DATA_BLOCK "JAMB_CLEANER_DB"	// DB 8
AUTHOR : Kamillas
VERSION : 0.1
  STRUCT
   JC_CAR_TRA_FWD_LS : BOOL ;	//JAMB CLEANER CARRIAGE TRAVEL FORWARD LIMIT SWITCH
   JC_CAR_TRA_RET_LS : BOOL ;	//JAMB CLEANER CARRIAGE TRAVEL RETRACT LIMIT SWITCH
   JC_VER_CLNR_UP_LS : BOOL ;	//JAMB CLEANER VERTICAL CLEANER UP LIMIT SWITCH
   JC_VER_CLNR_DN_LS : BOOL ;	//JAMB CLEANER VERTICAL CLEANER DOWN LIMIT SWITCH
   JC_VER_CLNR_HME_LS : BOOL ;	//JAMB CLEANER VERTICAL CLEANER HOME LIMIT SWITCH
   JC_CRA_TRA_FWD_STA_PB : BOOL ;	//JAMB CLEANER CARRIAGE TRAVEL FORWARD PUSH BUTTON
   JC_CRA_TRA_RET_STA_PB : BOOL ;	//JAMB CLEANER CARRIAGE TRAVEL RETRACT PUSH BUTTON
   JC_VC_UP_STA_PB : BOOL ;	//JAMB CLEANER VERTICAL CLEANER UP START PUSH BUTTON
   JC_VC_DN_STA_PB : BOOL ;	//JAMB CLEANER VERTICAL CLEANER DOWN START PUSH BUTTON
   JC_STP_PB : BOOL ;	//JAMB CLEANER OPERATIONS STOP PUSH BUTTON
   JC_VC_HME_STA_PB : BOOL ;	//JAMB CLEANER VERTICAL CLEANER HOME START PUSH BUTTON
   JC_CAR_TRA_FWD_CMD : BOOL ;	//JAMB CLEANER CARRIAGE TRAVEL FORWARD COMMAND
   JC_CAR_TRA_RET_CMD : BOOL ;	//JAMB CLEANER CARRIAGE TRAVEL RETRACT COMMAND
   JC_VC_UP_CMD : BOOL ;	//JAMB CLEANER VERTICAL CLEANER UP COMMAND
   JC_VC_DN_CMD : BOOL ;	//JAMB CLEANER VERTICAL CLEANER DOWN COMMAND
   JC_CAR_TRA_FWD_IND : BOOL ;	//JAMB CLEANER CARRIAGE TRAVEL FORWARD INDICATOR
   JC_CAR_TRA_RET_IND : BOOL ;	//JAMB CLEANER CARRIAGE TRAVEL RETRACT INDICATOR
   JC_VC_UP_IND : BOOL ;	//JAMB CLEANER VERTICAL CLEANER UP INDICATOR
   JC_VC_DN_IND : BOOL ;	//JAMB CLEANER VERTICAL CLEANER DOWN INDICATOR
   JC_VC_HME_IND : BOOL ;	//JAMB CLEANER VERTICAL CLEANER HOME INDIATOR
   CLN_OVN_JMB_STA_PB : BOOL ;	//CLEAN OVEN JAMB AUTO START PUSH BUTTON
   CLN_OVN_JMB_STP_PB : BOOL ;	//CLEAN OVEN JAMB AUTO STOP PUSH BUTTON
   CLN_OVN_JMB_IND : BOOL ;	//CLEAN OVEN JAMB AUTO INDICATOR
   JC_TRA_FWD_OP_CUT : BOOL ;	//JAMB CLEANER TRAVEL FORWARD OUTPUT CUT
   JC_TRA_FWD_OP_CUT_TMR : INT ;	//JAMB CLEANER TRAVEL FORWARD OUTPUT CUT TIMER
   JC_TRA_AUTO_FWD_OVR : BOOL ;	//JAMB CLEANER TRAVEL AUTO FORWARD OVER
   JC_TRA_AUTO_FWD_DEL : INT  := 3;	//JAMB CLEANER TRAVEL AUTO FORWARD OVER DELAY
   JC_TRA_AUTO_FWD_DEL_TMR : INT ;	//JAMB CLEANER TRAVEL AUTO FORWARD OVER DELAY TIMER
   JC_TRA_AUTO_FWD_SET : BOOL ;	//JAMB CLEANER AUTO TRAVEL FORWARD SET
   JC_TRA_RET_OP_CUT : BOOL ;	//JAMB CLEANER TRAVEL RETRACT OUTPUT CUT
   JC_TRA_RET_OP_CUT_TMR : INT ;	//JAMB CLEANER TRAVEL RETRACT OUTPUT CUT TIMER
   JC_TRA_AUTO_RET_OVR : BOOL ;	//JAMB CLEANER TRAVEL AUTO RETRACT OVER
   JC_TRA_AUTO_RET_DEL : INT  := 3;	//JAMB CLEANER TRAVEL AUTO RETRACT OVER DELAY
   JC_TRA_AUTO_RET_DEL_TMR : INT ;	//JAMB CLEANER TRAVEL AUTO RETRACT OVER DELAY TIMER
   JC_TRA_AUTO_RET_SET : BOOL ;	//JAMB CLEANER AUTO TRAVEL RETRACT SET
   JC_VC_FWD_OP_CUT : BOOL ;	//JAMB CLEANER VERTICAL CLEANER FORWARD OUTPUT CUT
   JC_VC_FWD_OP_CUT_TMR : INT ;	//JAMB CLEANER VERTICAL CLEANER FORWARD OUTPUT CUT TIMER
   JC_VC_AUTO_FWD_OVR : BOOL ;	//JAMB CLEANER VERTICAL CLEANER AUTO FORWARD OVER
   JC_VC_AUTO_FWD_DEL : INT  := 3;	//JAMB CLEANER VERTICAL CLEANER AUTO FORWARD OVER DELAY
   JC_VC_AUTO_FWD_DEL_TMR : INT ;	//JAMB CLEANER VERTICAL CLEANER AUTO FORWARD OVER DELAY TIMER
   JC_VC_AUTO_FWD_SET : BOOL ;	//JAMB CLEANER AUTO VERTICAL CLEANER FORWARD SET
   JC_VC_RET_OP_CUT : BOOL ;	//JAMB CLEANER VERTICAL CLEANER RETRACT OUTPUT CUT
   JC_VC_RET_OP_CUT_TMR : INT ;	//JAMB CLEANER VERTICAL CLEANER RETRACT OUTPUT CUT TIMER
   JC_VC_AUTO_RET_OVR : BOOL ;	//JAMB CLEANER VERTICAL CLEANER AUTO RETRACT OVER
   JC_VC_AUTO_RET_DEL : INT  := 3;	//JAMB CLEANER VERTICAL CLEANER AUTO RETRACT OVER DELAY
   JC_VC_AUTO_RET_DEL_TMR : INT ;	//JAMB CLEANER VERTICAL CLEANER AUTO RETRACT OVER DELAY TIMER
   JC_VC_AUTO_RET_SET : BOOL ;	//JAMB CLEANER AUTO VERTICAL CLEANER RETRACT SET
   JC_AUTO_SS : BOOL ;	//JAMB CLEANER AUTO MODE SELECTOR SWITCH
   JC_MAN_SS : BOOL ;	//JAMB CLEANER MANUAL MODE SELECTOR SWITCH
   JC_LOC_SS : BOOL ;	//JAMB CLEANER LOCAL MODE SELECTOR SWITCH
   JC_AUTO_STA_PB : BOOL ;	//JAMB CLEANER AUTO START PUSH BUTTON
   JC_ILK_BIT : BOOL ;	//JAMB CLEANER INTERLOCK BIT
   PULSE_1 : BOOL ;	//PULSE 1
   PULSE_2 : BOOL ;	//PULSE 2
   PULSE_3 : BOOL ;	//PULSE 3
   PULSE_4 : BOOL ;	//PULSE 4
   PULSE_5 : BOOL ;	//PULSE 5
   PULSE_6 : BOOL ;	//PULSE 6
   PULSE_7 : BOOL ;	//PULSE 7
   PULSE_8 : BOOL ;	//PULSE 8
   PULSE_9 : BOOL ;	//PULSE 9
   PULSE_10 : BOOL ;	//PULSE 10
   PULSE_11 : BOOL ;	//PULSE 11
   PULSE_12 : BOOL ;	//PULSE 12
   PULSE_13 : BOOL ;	//PULSE 13
   PULSE_14 : BOOL ;	//PULSE 14
   PULSE_15 : BOOL ;	//PULSE 15
   PULSE_16 : BOOL ;	//PULSE 16
   JC_HME_POS_BIT : BOOL ;	//JAMB CLEANER HOME POSITION BIT
   JC_VC_HME_OP_CUT : BOOL ;	//JAMB CLEANER VERTICAL CLEANER HOME OUTPUT CUT
   JC_VC_HME_OP_CUT_TMR : INT ;	//JAMB CLEANER VERTICAL CLEANER HOME OUTPUT CUT TIMER
   JC_VC_AUTO_HME_OVR : BOOL ;	//JAMB CLEANER VERTICAL CLEANER AUTO HOME OVER
   JC_VC_AUTO_HME_DEL : INT  := 3;	//JAMB CLEANER VERTICAL CLEANER AUTO HOME OVER DELAY
   JC_VC_AUTO_HME_DEL_TMR : INT ;	//JAMB CLEANER VERTICAL CLEANER AUTO HOME OVER DELAY TIMER
   JC_VC_AUTO_HME_SET : BOOL ;	//JAMB CLEANER AUTO VERTICAL CLEANER HOME SET
   JC_VC_HME_CMD : BOOL ;	//JAMB CLEANER AUTO VERTICAL CLEANER HOME COMMADN
   JC_AUTO_STA : BOOL ;	//JAMB CLEANER AUTO START BIT
   JC_CLN_OVN_JAMB_IND : BOOL ;	//CLEAN OVEN JAMB INDICATOR
   JC_CLN_OVN_JAMB_FIN : BOOL ;	//CLEAN OVEN JAMB FINISHED BIT
   JC_UP_DN_CNT : INT ;	//JAMB CLEANER UP/DOWN COUNT
   JC_UP_DN_CNT_SET : INT  := 3;	//JAMB CLEANER UP/DOWN COUNT SET POINT
   JC_UP_DN_CNT_OVR : BOOL ;	//JAMB CLEANER UP/DOWN COUNT OVER
  END_STRUCT ;	
BEGIN
   JC_TRA_AUTO_FWD_DEL := 3;
   JC_TRA_AUTO_RET_DEL := 3;
   JC_VC_AUTO_FWD_DEL := 3;
   JC_VC_AUTO_RET_DEL := 3;
   JC_VC_AUTO_HME_DEL := 3;
   JC_UP_DN_CNT_SET := 2;
END_DATA_BLOCK

DATA_BLOCK "GUIDE_CAGE_DB"	// DB 9
AUTHOR : Kamillas
VERSION : 0.1
  STRUCT
   GC_TRA_FWD_LS : BOOL ;	//GUIDE CAGE TRAVEL FORWARD LIMIT SWITCH
   GC_TRA_RET_LS : BOOL ;	//GUIDE CAGE TRAVEL RETRACT LIMIT SWITCH
   GC_AUTO_SS : BOOL ;	//GUIDE CAGE AUTO SELECTOR SWITCH
   GC_MAN_SS : BOOL ;	//GUIDE CAGE MANUAL SELECTOR SWITCH
   GC_TRA_FWD_STA_PB : BOOL ;	//GUIDE CAGE TRAVEL FORWARD START PUSH BUTTON
   GC_TRA_RET_STA_PB : BOOL ;	//GUIDE CAGE TRAVEL RETRACT START PUSH BUTTON
   GC_STP_PB : BOOL ;	//GUIDE CAGE AUTO STOP PUSH BUTTON
   GC_TRA_AUTO_STA_PB : BOOL ;	//GUIDE CAGE TRAVEL AUTO START PUSH BUTTON
   GC_TRA_AUTO_STP_PB : BOOL ;	//GUIDE CAGE TRAVEL AUTO STOP PUSH BUTTON
   GC_TRA_FWD_CMD : BOOL ;	//GUIDE CAGE TRAVEL FORWARD COMMAND
   GC_TRA_RET_CMD : BOOL ;	//GUIDE CAGE TRAVEL RETRACT COMMAND
   GC_TRA_FWD_IND : BOOL ;	//GUIDE CAGE TRAVEL FORWARD INDICATOR
   GC_TRA_RET_IND : BOOL ;	//GUIDE CAGE TRAVEL RETRACT INDICATOR
   GC_TRA_AUTO_IND : BOOL ;	//GUIDE CAGE AUTO OPERATION INDICATOR
   GC_TRA_FWD_OP_CUT : BOOL ;	//GUIDE CAGE TRAVEL FORWARD OUTPUT CUT
   GC_TRA_FWD_OP_CUT_TMR : INT ;	//GUIDE CAGE TRAVEL FORWARD OUTPUT CUT TIMER
   GC_TRA_AUTO_FWD_OVR : BOOL ;	//GUIDE CAGE TRAVEL AUTO FORWARD OVER
   GC_TRA_AUTO_FWD_DEL : INT  := 3;	//GUIDE CAGE TRAVEL AUTO FORWARD OVER DELAY
   GC_TRA_AUTO_FWD_DEL_TMR : INT ;	//GUIDE CAGE TRAVEL AUTO FORWARD OVER DELAY TIMER
   GC_TRA_AUTO_FWD_SET : BOOL ;	//GUIDE CAGE AUTO TRAVEL FORWARD SET
   GC_TRA_RET_OP_CUT : BOOL ;	//GUIDE CAGE TRAVEL RETRACT OUTPUT CUT
   GC_TRA_RET_OP_CUT_TMR : INT ;	//GUIDE CAGE TRAVEL RETRACT OUTPUT CUT TIMER
   GC_TRA_AUTO_RET_OVR : BOOL ;	//GUIDE CAGE TRAVEL AUTO RETRACT OVER
   GC_TRA_AUTO_RET_DEL : INT  := 3;	//GUIDE CAGE TRAVEL AUTO RETRACT OVER DELAY
   GC_TRA_AUTO_RET_DEL_TMR : INT ;	//GUIDE CAGE TRAVEL AUTO RETRACT OVER DELAY TIMER
   GC_TRA_AUTO_RET_SET : BOOL ;	//GUIDE CAGE AUTO TRAVEL RETRACT SET
   GC_AUTO_STA_PB : BOOL ;	//GUIDE CAGE AUTO START PUSH BUTTON
   GC_ILK_BIT : BOOL ;	//GUIDE CAGE INTERLOCK BIT
   PULSE_1 : BOOL ;	//PULSE 1
   PULSE_2 : BOOL ;	//PULSE 2
   PULSE_3 : BOOL ;	//PULSE 3
   PULSE_4 : BOOL ;	//PULSE 4
   PULSE_5 : BOOL ;	//PULSE 5
   PULSE_6 : BOOL ;	//PULSE 6
   PULSE_7 : BOOL ;	//PULSE 7
   PULSE_8 : BOOL ;	//PULSE 8
   PULSE_9 : BOOL ;	//PULSE 9
   PULSE_10 : BOOL ;	//PULSE 10
   PULSE_11 : BOOL ;	//PULSE 11
   PULSE_12 : BOOL ;	//PULSE 12
   PULSE_13 : BOOL ;	//PULSE 13
   PULSE_14 : BOOL ;	//PULSE 14
   PULSE_15 : BOOL ;	//PULSE 15
   PULSE_16 : BOOL ;	//PULSE 16
   GC_LOC_SS : BOOL ;	//GUIDE CAGE LOCAL SELECTOR SWITCH
   GC_AUTO_FWD_STA_BIT : BOOL ;	//GUIDE CAGE AUTO FORWARD START BIT
   GC_HME_POS_BIT : BOOL ;	//GUIDE CAGE HOME POSITION BIT
   GC_AUTO_RET_STA_BIT : BOOL ;	//GUIDE CAGE AUTO RETRACT START BIT
   GC_AUTO_OPER_FIN : BOOL ;	//GUIDE CAGE AUTO OPERATIONS FINISHED BIT
   GC_AUTO_OPER_IND : BOOL ;	//GUIDE CAGE AUTO OPERATIONS INDICATOR
   GC_PERM : BOOL ;	//GUIDE CAGE PERMISSION
  END_STRUCT ;	
BEGIN
   GC_TRA_AUTO_FWD_DEL := 3;
   GC_TRA_AUTO_RET_DEL := 3;
END_DATA_BLOCK

DATA_BLOCK "DOOR_CLEANER_MOTOR_DB"	// DB 10
AUTHOR : Kamillas
VERSION : 0.1
  STRUCT
   DC_MTR_RDY_FOR_STA : BOOL ;	//DOOR CLEANER READY FOR START
   DC_MTR_UP_RUN_FB : BOOL ;	//DOOR CLEANER UP RUNNING FEED BACK
   DC_MTR_OLR_TRIP : BOOL ;	//DOOR CLEANER OVER LOAD TRIP
   DC_MTR_DN_RUN_FB : BOOL ;	//DOOR CLEANER DOWN RUNNING FEED BACK
   DC_MTR_AUTO_SS : BOOL ;	//DOOR CLEANER AUTO SELECTOR SWITCH
   DC_MTR_MAN_SS : BOOL ;	//DOOR CLEANER MANUAL SELECTOR SWITCH
   DC_MTR_UP_STA_PB : BOOL ;	//DOOR CLEANER UP START PUSH BUTTON
   DC_MTR_DN_STA_PB : BOOL ;	//DOOR CLEANER DOWN START PUSH BUTTON
   DC_MTR_STP_PB : BOOL ;	//DOOR CLEANER STOP PUSH BUTTON
   DC_MTR_HME_PB : BOOL ;	//DOOR CLEANER HOME PUSH BUTTON
   DC_MTR_UP_LS : BOOL ;	//DOOR CLEANER UP LIMIT SWITCH
   DC_MTR_DN_LS : BOOL ;	//DOOR CLEANER DOWN LIMIT SWITCH
   DC_MTR_HME_LS : BOOL ;	//DOOR CLEANER HOME LIMIT SWITCH
   CLN_OVN_DR_STA_PB : BOOL ;	//CLEAN OVEN DOOR START PUSH BUTTON
   CLN_OVN_DR_STP_PB : BOOL ;	//CLEAN OVEN DOOR STOP PUSH BUTTON
   DC_MTR_UP_ON_CMD : BOOL ;	//DOOR CLEANER UP ON COMMAND
   DC_MTR_DN_ON_CMD : BOOL ;	//DOOR CLEANER DOWN ON COMMAND
   DC_MTR_UP_IND : BOOL ;	//DOOR CLEANER UP INDICATOR
   DC_MTR_DN_IND : BOOL ;	//DOOR CLEANER DOWN INDICATOR
   DC_MTR_HME_IND : BOOL ;	//DOOR CLEANER HOME INDICATOR
   CLN_OVN_DR_AUTO_IND : BOOL ;	//CLEAN OVEN DOOR AUTO INDICATOR
   DC_MTR_FLT : BOOL ;	//DOOR COMPRESSOR MOTOR FAULT
   DC_MTR_FLT_TMR : INT ;	//DOOR COMPRESSOR MOTOR FAULT TIMER
   DC_MTR_FLT_GEN_TIME : INT  := 3;	//DOOR COMPRESSOR MOTOR FAULT GEMERATION TIME
   PULSE_1 : BOOL ;	//PULSE 1
   PULSE_2 : BOOL ;	//PULSE 2
   PULSE_3 : BOOL ;	//PULSE 3
   PULSE_4 : BOOL ;	//PULSE 4
   PULSE_5 : BOOL ;	//PULSE 5
   PULSE_6 : BOOL ;	//PULSE 6
   PULSE_7 : BOOL ;	//PULSE 7
   PULSE_8 : BOOL ;	//PULSE 8
   DC_MTR_ILK_BIT : BOOL ;	//DOOR CLEANER MOTOR INTERLOCK BIT
   DC_MTR_AUTO_STA_BIT : BOOL ;	//DOOR CLEANER MOTOR AUTO START BIT
   DC_MTR_HME_POS_BIT : BOOL ;	//DOOR CLEANER MOTOR HOME POSITION BIT
   DC_MTR_UP_DN_CNT_OVR : BOOL ;	//DOOR CLEANER MOTOR UP DOWN COUNT OVER
   DC_MTR_UP_DN_CNT : INT ;	//DOOR CLEANER UP DOWN COUNT
   DC_MTR_UP_DN_CNT_SET : INT  := 1;	//DOOR CLEANER MOTOR UP DOWN COUNT SET POINT
   DC_MTR_LOC_SS : BOOL ;	//DOOR CLEANER MOTOR LOCAL SELECTOR SWITCH
   DC_MTR_HME_ON_CMD : BOOL ;	//DOOR CLEANER HOME ON COMMAND
   DC_MTR_CLN_OVN_DOOR_IND : BOOL ;	//DOOR CLEANER - CLEAN OVEN DOOR INDICATOR
   TRA_SLOW_FWD_OP_CUT : BOOL ;	//TRAVEL SLOW FORWARD OUTPUT CUT
   TRA_SLOW_FWD_FLT_TMR : INT ;	//TRAVEL SLOW FORWARD FAULT TIMER
   TRA_SLOW_FWD_FLT_GEN : INT  := 8;	//TRAVEL SLOW FORWARD FAULT GENERATION TIME
   TRA_SLOW_FWD_OP_CT_TM : INT ;	//TRAVEL SLOW FORWARD OUTPUT CUT TIMER
   TRA_SLOW_FWD_FLT : BOOL ;	//TRAVEL SLOW FORWARD FAULT
   TRA_SLOW_AUTO_FWD_OVR : BOOL ;	//TRAVEL SLOW AUTO FORWARD OVER
   TRA_SLOW_AUTO_FWD_DEL : INT  := 3;	//TRAVEL SLOW AUTO FORWARD OVER DELAY
   TRA_SLOW_ATO_FWD_DL_T : INT ;	//TRAVEL SLOW AUTO FORWARD OVER DELAY TIMER
   TRA_SLOW_RET_OP_CUT : BOOL ;	//TRAVEL SLOW RETRACT OUTPUT CUT
   TRA_SLOW_RET_FLT_TMR : INT ;	//TRAVEL SLOW RETRACT FAULT TIMER
   TRA_SLOW_RET_FLT_GEN : INT  := 8;	//TRAVEL SLOW RETRACT FAULT GENERATION TIME
   TRA_SLOW_RET_OP_CT_TM : INT ;	//TRAVEL SLOW RETRACT OUTPUT CUT TIMER
   TRA_SLOW_RET_FLT : BOOL ;	//TRAVEL SLOW RETRACT FAULT
   TRA_SLOW_AUTO_RET_OVR : BOOL ;	//TRAVEL SLOW AUTO RETRACT OVER
   TRA_SLOW_AUTO_RET_DEL : INT  := 3;	//TRAVEL SLOW AUTO RETRACT OVER DELAY
   TRA_SLOW_ATO_RET_DL_T : INT ;	//TRAVEL SLOW AUTO RETRACT OVER DELAY TIMER
   TRA_NOR_FWD_OP_CUT : BOOL ;	//TRAVEL NORMAL FORWARD OUTPUT CUT
   TRA_NOR_FWD_FLT_TMR : INT ;	//TRAVEL NORMAL FORWARD FAULT TIMER
   TRA_NOR_FWD_FLT_GEN : INT  := 8;	//TRAVEL NORMAL FORWARD FAULT GENERATION TIME
   TRA_NOR_FWD_OP_CT_TM : INT ;	//TRAVEL NORMAL FORWARD OUTPUT CUT TIMER
   TRA_NOR_FWD_FLT : BOOL ;	//TRAVEL NORMAL FORWARD FAULT
   TRA_NOR_AUTO_FWD_OVR : BOOL ;	//TRAVEL NORMAL AUTO FORWARD OVER
   TRA_NOR_AUTO_FWD_DEL : INT  := 3;	//TRAVEL NORMAL AUTO FORWARD OVER DELAY
   TRA_NOR_ATO_FWD_DL_T : INT ;	//TRAVEL NORMAL AUTO FORWARD OVER DELAY TIMER
   TRA_NOR_RET_OP_CUT : BOOL ;	//TRAVEL NORMAL RETRACT OUTPUT CUT
   TRA_NOR_RET_FLT_TMR : INT ;	//TRAVEL NORMAL RETRACT FAULT TIMER
   TRA_NOR_RET_FLT_GEN : INT  := 8;	//TRAVEL NORMAL RETRACT FAULT GENERATION TIME
   TRA_NOR_RET_OP_CT_TM : INT ;	//TRAVEL NORMAL RETRACT OUTPUT CUT TIMER
   TRA_NOR_RET_FLT : BOOL ;	//TRAVEL NORMAL RETRACT FAULT
   TRA_NOR_AUTO_RET_OVR : BOOL ;	//TRAVEL NORMAL AUTO RETRACT OVER
   TRA_NOR_AUTO_RET_DEL : INT  := 3;	//TRAVEL NORMAL AUTO RETRACT OVER DELAY
   TRA_NOR_ATO_RET_DL_T : INT ;	//TRAVEL NORMAL AUTO RETRACT OVER DELAY TIMER
   TRA_SLOW_FWD_CMD : BOOL ;	//TRAVEL SLOW FORWARD COMMAND
   TRA_SLOW_RET_CMD : BOOL ;	//TRAVEL SLOW RETRACT COMMAND
   TRA_NOR_FWD_CMD : BOOL ;	//TRAVEL NORMAL FORWARD COMMAND
   TRA_NOR_RET_CMD : BOOL ;	//TRAVEL NORMAL RETRACT COMMAND
   TRA_RELIVE_CMD : BOOL ;	//TRAVEL RELIVE COOMMAND
   TRA_AUTO_FWD_CLN_POS_SET : BOOL ;	//TRAVEL AUTO FORWARD TO CLEANING POSITION SET
   TRA_AUTO_RET_SET : BOOL ;	//TRAVEL AUTO RETRACT SET
   TRA_CLN_POS_LS : BOOL ;	//TRAVEL CLEANING POSTION LIMIT SWITCH
   PULSE_9 : BOOL ;	//PULSE 9
   PULSE_10 : BOOL ;	//PULSE 10
   PULSE_11 : BOOL ;	//PULSE 11
   PULSE_12 : BOOL ;	//PULSE 12
   PULSE_13 : BOOL ;	//PULSE 13
   PULSE_14 : BOOL ;	//PULSE 14
   PULSE_15 : BOOL ;	//PULSE 15
   PULSE_16 : BOOL ;	//PULSE 16
   DC_MTR_HME_SET : BOOL ;	//TRAVEL AUTO HOME SET
   DC_MTR_AUTO_OPER_FIN : BOOL ;	//DOOR CLEANER MOTOR AUTO OPERATIONS FINISHED
   DC_AUTO_STOPPED : BOOL ;	//DOOR CLEANER OPERATIONS STOPED WHILE IN AUTO OPERATION
   DC_MTR_UP_LS_HOLD : BOOL ;	//UP LIMIT SWITCH HOLDING
   DC_MTR_DN_LS_HOLD : BOOL ;	//DOWN LIMIT SWITCH HOLDING
   DC_MTR_HME_LS_HOLD : BOOL ;	//HOME LIMIT SWITCH HOLDING
  END_STRUCT ;	
BEGIN
   DC_MTR_FLT_GEN_TIME := 3;
   DC_MTR_UP_DN_CNT_SET := 1;
   TRA_SLOW_FWD_FLT_GEN := 8;
   TRA_SLOW_AUTO_FWD_DEL := 3;
   TRA_SLOW_RET_FLT_GEN := 8;
   TRA_SLOW_AUTO_RET_DEL := 3;
   TRA_NOR_FWD_FLT_GEN := 8;
   TRA_NOR_AUTO_FWD_DEL := 3;
   TRA_NOR_RET_FLT_GEN := 8;
   TRA_NOR_AUTO_RET_DEL := 3;
END_DATA_BLOCK

DATA_BLOCK "WIN_CC_DB"	// DB 11
AUTHOR : Kamilas
VERSION : 0.1
  STRUCT
   MAIN_PWR_ON_PB : BOOL ;	//MAIN POWER ON PUSH BUTTON
   MAIN_PWR_OFF_PB : BOOL ;	//MAIN POWER OFF PUSH BUTTON
   MP_LAMP_TEST_PB : BOOL ;	//MAIN POWER LAMP TEST PUSH BUTTON
   MP_ALARM_ACK_PB : BOOL ;	//MAIN POWER ALARM ACKNOWLEDGE PUSH BUTTON
   CTRL_SELECTION_CD : BOOL ;	//CONTROL SELECTRION CD
   ALL_MECH_QUICK_STP : BOOL ;	//ALL MECHANICAL QUICK STOP
   REP_MAN_SS : BOOL ;	//REPAIR MANUAL SELECTION
   SEMI_AUTO_SS : BOOL ;	//SEMI AUTO SELECTION
   PUMP_1_RDY_FOR_STA : BOOL ;	//PUMP 1 READY FOR START
   PUMP_2_RDY_FOR_STA : BOOL ;	//PUMP 2 READY FOR START
   CIR_PUMP_RDY_FOR_STA : BOOL ;	//CIRCULATION PUMP READY FOR START
   COLR_FAN_RDY_FOR_STA : BOOL ;	//COOLER FAN READY FOR START
   CD_LCS_SS : BOOL ;	//CONTROL DESK / LOCAL CONTROL SELECTOR SWITCH
   HY_PUMP_1_2_SS : BOOL ;	//PUMP 1 OR 2 SELECTOR SWITCH
   HY_PUMP_1_STA_PB : BOOL ;	//PUMP 1 START PUSH BUTTON
   HY_PUMP_1_STP_PB : BOOL ;	//PUMP 1 STOP PUSH BUTTON
   HY_PUMP_2_STA_PB : BOOL ;	//PUMP 2 START PUSH BUTTON
   HY_PUMP_2_STP_PB : BOOL ;	//PUMP 2 STOP PUSH BUTTON
   HY_PUMP_1_2_SS_LCS : BOOL ;	//PUMP 1 OR 2 SELECTOR SWITCH LCS
   HY_PUMP_1_STA_PB_LCS : BOOL ;	//PUMP 1 START PUSH BUTTON LCS
   HY_PUMP_1_STP_PB_LCS : BOOL ;	//PUMP 1 STOP PUSH BUTTON LCS
   HY_PUMP_2_STA_PB_LCS : BOOL ;	//PUMP 2 START PUSH BUTTON LCS
   HY_PUMP_2_STP_PB_LCS : BOOL ;	//PUMP 2 STOP PUSH BUTTON LCS
   HY_CIR_PUMP_STA_PB_LCS : BOOL ;	//CIRCULATION PUMP START PUSH BUTTON LCS
   HY_CIR_PUMP_STP_PB_LCS : BOOL ;	//CIRCULATION PUMP STOP PUSH BUTTON LCS
   HY_COLR_FAN_STA_PB_LCS : BOOL ;	//COOLER FAN START PUSH BUTTON LCS
   HY_COLR_FAN_STP_PB_LCS : BOOL ;	//COOLER FAN STOP PUSH BUTTON LCS
   TRA_DRV_1_BRK_RDY_FOR_ST : BOOL ;	//TRAVEL GROUP 1 BREAK READY FOR START
   TRA_DRV_2_BRK_RDY_FOR_ST : BOOL ;	//TRAVEL GROUP 2 BREAK READY FOR START
   TRA_MODE_AUTO_MAN_SS : BOOL ;	//TRAVEL MODE AUTO/MANUAL BUTTON
   TRA_DRV_1_PROF_HARD_SS : BOOL ;	//TRAVEL DRIVE 1 PROFIBUS/HARD WIRE SELECTRO SWITCH
   TRA_DRV_1_RDY_FOR_STA : BOOL ;	//TRAVEL DRIVE 1 READY FOR START
   TRA_DRV_2_PROF_HARD_SS : BOOL ;	//TRAVEL DRIVE 2 PROFIBUS/HARD WIRE SELECTRO SWITCH
   TRA_DRV_2_RDY_FOR_STA : BOOL ;	//TRAVEL DRIVE 2 READY FOR START
   AC_MTR_RDY_FOR_STA : BOOL ;	//AIR COMPRESSOR MOTOR READY FOR START
   AC_MTR_STA_PB : BOOL ;	//AIR COMPRESSOR MOTOR START PUSH BUTTON
   AC_MTR_STP_PB : BOOL ;	//AIR COMPRESSOR MOTOR STOP PUSH BUTTON
   IDF_DRV_RDY_FOR_STA : BOOL ;	//ID FAN DRIVE READY FOR START
   WTR_PMP_MTR_RDY_FOR_STA : BOOL ;	//WATER PUMP MOTOR READY FOR START
   HOOD_STA_PB : BOOL ;	//HOOD START PUSH BUTTON
   HOOD_STP_PB : BOOL ;	//HOOD STOP PUSH BUTTON
   IDF_DRV_LS_HS_SEL : BOOL ;	//ID FAN DRIVE LOW SPEED/HIGH SPEED SELECTION
   DE_DOOR_EXT_LOC_SS : BOOL ;	//DOOR EXTRACTOR LOCAL SELECTOR SWITCH
   DE_DOOR_EXT_MAN_SS : BOOL ;	//DOOR EXTRACTOR MANUAL SELECTOR SWITCH
   DE_DOOR_EXT_AUTO_SS : BOOL ;	//DOOR EXTRACTOR AUTO SELECTOR SWITCH
   DE_DOOR_EXT_STP_PB : BOOL ;	//DOOR EXTRACTOR STOP PUSH BUTTON
   DE_SLEW_FWD_STA_PB : BOOL ;	//SLEW FORWARD START PUSH BUTTON
   DE_SLEW_RET_STA_PB : BOOL ;	//SLEW RETRACT START
   DE_VER_COMP_FWD_STA_PB : BOOL ;	//VERTICAL COMPENSATION FORWARD START PUSH BUTTON
   DE_VER_COMP_RET_STA_PB : BOOL ;	//VERTICAL COMPENSATION RETRACT START PUSH BUTTON
   DE_TRA_FWD_STA_PB : BOOL ;	//TRAVEL FORWARD START PUSH BUTTON
   DE_TRA_RET_STA_PB : BOOL ;	//TRAVEL RETRACT START PUSH BUTTON
   MAIN_STK_UP_STA_PB : BOOL ;	//MAIN STROKE UP START PUSH BUTTON
   MAIN_STK_DN_PB : BOOL ;	//MAIN STROKE DOWN START PUSH BUTTON
   FIN_STK_UP_STA_PB : BOOL ;	//FINAL STROKE UP START PUSH BUTTON
   FIN_STK_DN_PB : BOOL ;	//FINAL STROKE DOWN START PUSH BUTTON
   PRE_STK_UP_STA_PB : BOOL ;	//PRE STROKE UP START PUSH BUTTON
   PRE_STK_UP_DN_PB : BOOL ;	//PRE STROKE DOWN START PUSH BUTTON
   DR_SPNG_LK_STA_PB : BOOL ;	//DOOR SPRING PRESSURE START PUSH BUTTON
   DR_SPNG_UNLK_STA_PB : BOOL ;	//DOOR SPRING PRESSURE RELEASE START PUSH BUTTON
   DR_LCH_TURN_UP_PB : BOOL ;	//DOOR LATCH TURNING LOCK PUSH BUTTON
   DR_LCH_TURN_DN_PB : BOOL ;	//DOOR LATCH TURNING UNLOCK PUSH BUTTON
   JC_CRA_TRA_FWD_STA_PB : BOOL ;	//JAMB CLEANER CARRIAGE TRAVEL FORWARD PUSH BUTTON
   JC_CRA_TRA_RET_STA_PB : BOOL ;	//JAMB CLEANER CARRIAGE TRAVEL RETRACT PUSH BUTTON
   JC_VC_UP_STA_PB : BOOL ;	//JAMB CLEANER VERTICAL CLEANER UP START PUSH BUTTON
   JC_VC_DN_STA_PB : BOOL ;	//JAMB CLEANER VERTICAL CLEANER DOWN START PUSH BUTTON
   JC_STP_PB : BOOL ;	//JAMB CLEANER OPERATIONS STOP PUSH BUTTON
   JC_VC_HME_STA_PB : BOOL ;	//JAMB CLEANER VERTICAL CLEANER HOME START PUSH BUTTON
   CLN_OVN_JMB_STA_PB : BOOL ;	//CLEAN OVEN JAMB AUTO START PUSH BUTTON
   CLN_OVN_JMB_STP_PB : BOOL ;	//CLEAN OVEN JAMB AUTO STOP PUSH BUTTON
   JC_AUTO_SS : BOOL ;	//JAMB CLEANER AUTO MODE SELECTOR SWITCH
   JC_MAN_SS : BOOL ;	//JAMB CLEANER MANUAL MODE SELECTOR SWITCH
   JC_LOC_SS : BOOL ;	//JAMB CLEANER LOCAL MODE SELECTOR SWITCH
   JC_AUTO_STA_PB : BOOL ;	//JAMB CLEANER AUTO START PUSH BUTTON
   GC_AUTO_SS : BOOL ;	//GUIDE CAGE AUTO SELECTOR SWITCH
   GC_MAN_SS : BOOL ;	//GUIDE CAGE MANUAL SELECTOR SWITCH
   GC_TRA_FWD_STA_PB : BOOL ;	//GUIDE CAGE TRAVEL FORWARD START PUSH BUTTON
   GC_TRA_RET_STA_PB : BOOL ;	//GUIDE CAGE TRAVEL RETRACT START PUSH BUTTON
   GC_STP_PB : BOOL ;	//GUIDE CAGE AUTO STOP PUSH BUTTON
   GC_TRA_AUTO_STA_PB : BOOL ;	//GUIDE CAGE TRAVEL AUTO START PUSH BUTTON
   GC_TRA_AUTO_STP_PB : BOOL ;	//GUIDE CAGE TRAVEL AUTO STOP PUSH BUTTON
   GC_AUTO_STA_PB : BOOL ;	//GUIDE CAGE AUTO START PUSH BUTTON
   DC_MTR_RDY_FOR_STA : BOOL ;	//DOOR CLEANER READY FOR START
   DC_MTR_AUTO_SS : BOOL ;	//DOOR CLEANER AUTO SELECTOR SWITCH
   DC_MTR_MAN_SS : BOOL ;	//DOOR CLEANER MANUAL SELECTOR SWITCH
   DC_MTR_UP_STA_PB : BOOL ;	//DOOR CLEANER UP START PUSH BUTTON
   DC_MTR_DN_STA_PB : BOOL ;	//DOOR CLEANER DOWN START PUSH BUTTON
   DC_MTR_STP_PB : BOOL ;	//DOOR CLEANER STOP PUSH BUTTON
   DC_MTR_HME_PB : BOOL ;	//DOOR CLEANER HOME PUSH BUTTON
   CLN_OVN_DR_STA_PB : BOOL ;	//CLEAN OVEN DOOR START PUSH BUTTON
   CLN_OVN_DR_STP_PB : BOOL ;	//CLEAN OVEN DOOR STOP PUSH BUTTON
   DC_MTR_LOC_SS : BOOL ;	//DOOR CLEANER MOTOR LOCAL SELECTOR SWITCH
   SP_STP_PB : BOOL ;	//SERVICE PLATFORM STOP PUSH BUTTON
   SP_STA_PB : BOOL ;	//SERVICE PLATFORM START PUSH BUTTON
   EMG_ACCM_STA_PB_LCS : BOOL ;	//EMERGENCY ACCUMULATOR START PUSH BUTTON LCS
   EMG_ACCM_STP_PB_LCS : BOOL ;	//EMERGENCY ACCUMULATOR STOP PUSH BUTTON LCS
   EXT_OVN_DOR_STA_PB : BOOL ;	//EXTRACT OVEN DOOR START PUSH BUTTON
   EXT_RPL_FUNC_STP_PB : BOOL ;	//EXTRACT AND REPLACE FUNCTIONAL STOP PUSH BUTTON
   RPL_OVN_DOR_STA_PB : BOOL ;	//REPLACE OVEN DOOR START PUSH BUTTON
   ALL_OPER_IN_OPER_MODE : BOOL ;	//ALL OPERATION IN OPERATION MODE
   ALL_OPER_IN_REP_MODE : BOOL ;	//ALL OPERATION IN REPAIR MODE
   SP_TRA_FWD_STA_PB : BOOL ;	//SERVICE PLATFORM TRAVEL FORWARD START PUSH BUTTON
   SP_TRA_REV_STA_PB : BOOL ;	//SERVICE PLATFORM TRAVEL REVERSE START PUSH BUTTON
   EMERGENCY_STOP : BOOL ;	//EMERGENCY STOP
   HY_LAMP_TEST : BOOL ;	//HYDRALIC SYSTEM LAMP PUSH BUTTON
   SP_AUTO_STP_PB : BOOL ;	//SERVICE PLATFORM AUTO STOP PUSH BUTTON
   SP_TRA_AUTO_STA_PB : BOOL ;	//SERVICE PLATFORM TRAVEL AUTO START PUSH BUTTON
   SP_TRA_AUTO_STP_PB : BOOL ;	//SERVICE PLATFORM TRAVEL AUTO STOP PUSH BUTTON
   SP_AUTO_STA_PB : BOOL ;	//SERVICE PLATFORM AUTO START PUSH BUTTON
   SP_AUTO_SS : BOOL ;	//SERVICE PLATFORM AUTO MODE SELECTOR SWITCH
   SP_MAN_SS : BOOL ;	//SERVICE PLATFORM MANUAL MODE SELECTOR SWITCH
   MAIN_PWR_RDY_FOR_ON : BOOL ;	//MAIN POWER READY FOR ON
   MAIN_PWR_ON_FB : BOOL ;	//MAIN POWER ON FEED BACK
   CTRL_PWR_ON_FB : BOOL ;	//CONTROL POWER ON FEEDBACK
   PUMP_1_RUN_FB : BOOL ;	//PUMP 1 RUNNING FEEDBACK
   PUMP_1_OVR_LD_TRIP : BOOL ;	//PUMP 1 OVER LOAD TRIPPED
   PUMP_2_RUN_FB : BOOL ;	//PUMP 2 RUNNING FEEDBACK
   PUMP_2_OVR_LD_TRIP : BOOL ;	//PUMP 2 OVER LOAD TRIPPED
   CIR_PUMP_RUN_FB : BOOL ;	//CIRCULATION PUMP RUNNING FEEDBACK
   CIR_PUMP_OVR_LD_TRIP : BOOL ;	//CIRCULATION PUMP OVER LOAD TRIPPED
   COLR_FAN_RUN_FB : BOOL ;	//COOLER FAN RUNNING FEEDBACK
   COLR_FAN_OVR_LD_TRIP : BOOL ;	//COOLER FAN OVER LOAD TRIPPED
   SHT_OF_VLV_LIN_1_FUL_OPN : BOOL ;	//SHUT OFF VALVE IN LINE 1 - FULLY OPEN
   SHT_OF_VLV_LIN_2_FUL_OPN : BOOL ;	//SHUT OFF VALVE IN LINE 2 - FULLY OPEN
   LOW_OIL_TEMP : BOOL ;	//LOW OIL TEMPERATURE - THERMOSTAT
   HIGH_OIL_TEMP : BOOL ;	//HIGH OIL TEMPERATURE - THERMOSTAT
   MAX_OIL_TEMP : BOOL ;	//MAXIMUM OIL TEMPERATURE - THERMOSTAT
   LOW_OIL_LEVEL : BOOL ;	//LOW OIL LEVEL - FLOAT SWITCH
   MIN_OIL_LEVEL : BOOL ;	//MINIMUM OIL LEVEL - FLOAT SWITCH
   RET_LIN_FLTR_CKD : BOOL ;	//RETURN LINE FILTER CHOKED
   TRA_DRV_1_ON_FB : BOOL ;	//TRAVEL DRIVE 1 ON FEEDBACK
   TRA_DRV_1_TRP_FB : BOOL ;	//TRAVEL DRIVE 1 TRIP FEEDBACK
   SLEW_SLOW_FWD_LS : BOOL ;	//SLEW SLOW FORWARD LIMIT SWITCH
   SLEW_SLOW_RET_LS : BOOL ;	//SLEW SLOW RETRACT LIMIT SWITCH
   SLEW_NOR_FWD_LS : BOOL ;	//SLEW NORMAL FORWARD LIMIT SWITCH
   SLEW_NOR_RET_LS : BOOL ;	//SLEW NORMAL RETRACT LIMIT SWITCH
   TRA_SLOW_FWD_LS : BOOL ;	//TRAVEL SLOW FORWARD LIMIT  SWITCH
   TRA_SLOW_RET_LS : BOOL ;	//TRAVEL SLOW RETRACT LIMIT  SWITCH
   TRA_FWD_LS : BOOL ;	//TRAVEL FORWARD LIMIT SWIITCH
   TRA_RET_LS : BOOL ;	//TRAVEL RETRACT LIMIT SWIITCH
   FOR_LS_TRAVEL : BOOL ;	//FORWARD LIMIT SWITCH TRAVEL
   DOOR_ON_HOOK_LS : BOOL ;	//DOOR ON HOOK LIMITSWTCH
   JC_CAR_TRA_FWD_LS : BOOL ;	//JAMB CLEANER CARRIAGE TRAVEL FORWARD LIMIT SWITCH
   JC_CAR_TRA_RET_LS : BOOL ;	//JAMB CLEANER CARRIAGE TRAVEL RETRACT LIMIT SWITCH
   JC_VER_CLNR_UP_LS : BOOL ;	//JAMB CLEANER VERTICAL CLEANER UP LIMIT SWITCH
   JC_VER_CLNR_DN_LS : BOOL ;	//JAMB CLEANER VERTICAL CLEANER DOWN LIMIT SWITCH
   JC_VER_CLNR_HME_LS : BOOL ;	//JAMB CLEANER VERTICAL CLEANER HOME LIMIT SWITCH
   DC_MTR_UP_LS : BOOL ;	//DOOR CLEANER UP LIMIT SWITCH
   DC_MTR_DN_LS : BOOL ;	//DOOR CLEANER DOWN LIMIT SWITCH
   AC_MTR_RUN_FB : BOOL ;	//AIR COMPRESSOR MOTOR RUN FEED BACK
   AC_MTR_OLR_TRIP_FB : BOOL ;	//AIR COMPRESSOR MOTOR TRIP FEED BACK
   GC_TRA_FWD_LS : BOOL ;	//GUIDE CAGE TRAVEL FORWARD LIMIT SWITCH
   GC_TRA_RET_LS : BOOL ;	//GUIDE CAGE TRAVEL RETRACT LIMIT SWITCH
   TRA_JOY_STK_FWD_POS : BOOL ;	//TRAVEL JOY STICK FOWRWARD POSITION
   TRA_JOY_STK_REV_POS : BOOL ;	//TRAVEL JOY DEAD REVERSE POSITION
   TRA_JOY_STK_HME_POS : BOOL ;	//TRAVEL JOY STICK HOME POSITION
   TRA_JOY_STK_DED_MAN_BTN : BOOL ;	//TRAVEL JOY DEAD MAN BUTTON
   TRA_DRV_2_ON_FB : BOOL ;	//TRAVEL DRIVE 2 ON FEEDBACK
   TRA_DRV_2_TRP_FB : BOOL ;	//TRAVEL DRIVE 2 TRIP FEEDBACK
   DC_MTR_HME_LS : BOOL ;	//DOOR CLEANER HOME LIMIT SWITCH
   LAMP_TEST_PB : BOOL ;	//LAMP TEST PUSH BUTTON
   q : BOOL ;
   W : BOOL ;
   E : BOOL ;
   R : BOOL ;
   T : BOOL ;
   Y : BOOL ;
   U : BOOL ;
   REPR_OPER_MODE_SS : BOOL ;
   q1 : BOOL ;
   W1 : BOOL ;
   E1 : BOOL ;
   R1 : BOOL ;
   T1 : BOOL ;
   Y1 : BOOL ;
   U1 : BOOL ;
   TRAV_AUTO_MAN_SS : BOOL ;
   q11 : BOOL ;
   W11 : BOOL ;
   E11 : BOOL ;
   R11 : BOOL ;
   T11 : BOOL ;
   Y11 : BOOL ;
   U11 : BOOL ;
   SP_AUTO_MAN_SS : BOOL ;
   q111 : BOOL ;
   W111 : BOOL ;
   E111 : BOOL ;
   R111 : BOOL ;
   T111 : BOOL ;
   Y111 : BOOL ;
   U111 : BOOL ;
   GC_AUTO_MAN_SS : BOOL ;
   q1111 : BOOL ;
   W1111 : BOOL ;
   E1111 : BOOL ;
   R1111 : BOOL ;
   T1111 : BOOL ;
   Y1111 : BOOL ;
   U1111 : BOOL ;
   DC_AUTO_MAN_SS : BOOL ;
   q11111 : BOOL ;
   W11111 : BOOL ;
   E11111 : BOOL ;
   R11111 : BOOL ;
   T11111 : BOOL ;
   Y11111 : BOOL ;
   U11111 : BOOL ;
   JC_AUTO_MAN_SS : BOOL ;
   q111111 : BOOL ;
   W111111 : BOOL ;
   E111111 : BOOL ;
   R111111 : BOOL ;
   T111111 : BOOL ;
   Y111111 : BOOL ;
   U111111 : BOOL ;
   DE_AUTO_MAN_SS : BOOL ;
   q1111111 : BOOL ;
   W1111111 : BOOL ;
   E1111111 : BOOL ;
   R1111111 : BOOL ;
   T1111111 : BOOL ;
   Y1111111 : BOOL ;
   U1111111 : BOOL ;
   PUMP_CD_LCS_SS : BOOL ;
   q11111111 : BOOL ;
   W11111111 : BOOL ;
   E11111111 : BOOL ;
   R11111111 : BOOL ;
   T11111111 : BOOL ;
   Y11111111 : BOOL ;
   U11111111 : BOOL ;
   PUMP_1_2_SS : BOOL ;
   A : BOOL ;
   S : BOOL ;
   D : BOOL ;
   F : BOOL ;
   G : BOOL ;
   H : BOOL ;
   J : BOOL ;
   ID_FAN_HS_LS_SEL : BOOL ;
   A1 : BOOL ;
   S1 : BOOL ;
   D1 : BOOL ;
   F1 : BOOL ;
   G1 : BOOL ;
   H1 : BOOL ;
   J1 : BOOL ;
   JMB_CLN_HME_STA_PB : BOOL ;
  END_STRUCT ;	
BEGIN
END_DATA_BLOCK

DATA_BLOCK "CMD_FROM_TATA"	// DB 12
VERSION : 0.1
  STRUCT
   GC_OnBord_STATUS_BIT : STRUCT
    PUSH_PERM : BOOL ;	//Pushing interlock OK
    GC_LT_MODE : BOOL ;	//Long travel in auto or in man
    GC_TRAVEL_FWD : BOOL ;	//FWD over profibus
    GC_TRAVEL_REV : BOOL ;	//REV over profibus
    GC_TRAVEL_START : BOOL ;	//START over profibus
    GC_TRAVEL_STOP : BOOL ;	//STOP  over profibus
    SpareBit_1 : BOOL ;
    HOOD_SYS_ON_CMD : BOOL ;	//HOOD SYSTEM ON COMMAND
    GUIDE_CAGE_PERM : BOOL ;	//GUIDE CAGE PERMISSION
    SpareBit_4 : BOOL ;
    SpareBit_5 : BOOL ;
    SpareBit_6 : BOOL ;
    SpareBit_7 : BOOL ;
    SpareBit_8 : BOOL ;
    SpareBit_9 : BOOL ;
    SpareBit_10 : BOOL ;
    GC_SPEED_REF : INT ;	//Reserve for LT motion (spd_ref) over profibus
    SATA : ARRAY  [1 .. 7 ] OF INT ;
   END_STRUCT ;
  END_STRUCT ;	
BEGIN
END_DATA_BLOCK

DATA_BLOCK "FB_TO_TATA"	// DB 13
VERSION : 0.1
  STRUCT
   GC_MACHINE_STATUS_BIT : STRUCT
    COKE_SIDE_DOOR_CL : BOOL ;
    COKE_SIDE_DOOR_OP : BOOL ;
    GC_DRV_STATUS : BOOL ;
    GC_DRV_FWD : BOOL ;
    GC_DRV_REV : BOOL ;
    GC_PERM : BOOL ;
    GC_STATUS : BOOL ;
    SpareBit_2 : BOOL ;
    SpareBit_3 : BOOL ;
    TRA_AUTO_MAN_SELECT : BOOL ;	//TRAVEL AUTO MANUAL SELECTION
    SP_TRA_FWD_LS_REACH : BOOL ;	//SERVICE PLATFORM TRAVEL FORWARD REACHED
    SpareBit_6 : BOOL ;
    SpareBit_7 : BOOL ;
    SpareBit_8 : BOOL ;
    SpareBit_9 : BOOL ;
    SpareBit_10 : BOOL ;
    GC_SPEED : REAL ;
    Spare_Int0 : INT ;
    Spare_Int1 : INT ;
    SATA : ARRAY  [1 .. 4 ] OF INT ;
   END_STRUCT ;
  END_STRUCT ;	
BEGIN
END_DATA_BLOCK

DATA_BLOCK "TATA_COMMUNICATION_DB"	// DB 14
VERSION : 0.1
  STRUCT
   TATA_DATA_READ_ERROR : INT ;	//TATA PLC DATA READ ERROR
   TATA_DATA_WRITE_ERROR : INT ;	//TATA PLC DATA WRITE ERROR
   DR_OPN_LCH_TIMER : INT ;	//DOOR OPEN BIT LATCH TIMER
   DR_OPN_LCH_TIME : INT  := 5;	//DOOR OPEN BIT LATCH TIME
   DR_CLS_LCH_TIMER : INT ;	//DOOR CLOSE BIT LATCH TIMER
   DR_CLS_LCH_TIME : INT  := 5;	//DOOR CLOSE BIT LATCH TIME
   PUSLE_1 : BOOL ;	//PUSLE 1
   PUSLE_2 : BOOL ;	//PUSLE 2
   PUSLE_3 : BOOL ;	//PUSLE 3
   PUSLE_4 : BOOL ;	//PUSLE 4
   PUSLE_5 : BOOL ;	//PUSLE 5
   PUSLE_6 : BOOL ;	//PUSLE 6
   PUSLE_7 : BOOL ;	//PUSLE 7
   PUSLE_8 : BOOL ;	//PUSLE 8
  END_STRUCT ;	
BEGIN
   DR_OPN_LCH_TIME := 5;
   DR_CLS_LCH_TIME := 5;
END_DATA_BLOCK

ORGANIZATION_BLOCK "MAIN_PROGRAM"	// OB 1
TITLE = "Main Program Sweep (Cycle)"
AUTHOR : Kamillas
VERSION : 0.1
VAR_TEMP
  OB1_EV_CLASS : BYTE ;	//Bits 0-3 = 1 (Coming event), Bits 4-7 = 1 (Event class 1)
  OB1_SCAN_1 : BYTE ;	//1 (Cold restart scan 1 of OB 1), 3 (Scan 2-n of OB 1)
  OB1_PRIORITY : BYTE ;	//Priority of OB Execution
  OB1_OB_NUMBR : BYTE ;	//1 (Organization block 1, OB1)
  OB1_RESERVED_1 : BYTE ;	//Reserved for system
  OB1_RESERVED_2 : BYTE ;	//Reserved for system
  OB1_PREV_CYCLE : INT ;	//Cycle time of previous OB1 scan (milliseconds)
  OB1_MIN_CYCLE : INT ;	//Minimum cycle time of OB1 (milliseconds)
  OB1_MAX_CYCLE : INT ;	//Maximum cycle time of OB1 (milliseconds)
  OB1_DATE_TIME : DATE_AND_TIME ;	//Date and time OB1 started
END_VAR
BEGIN
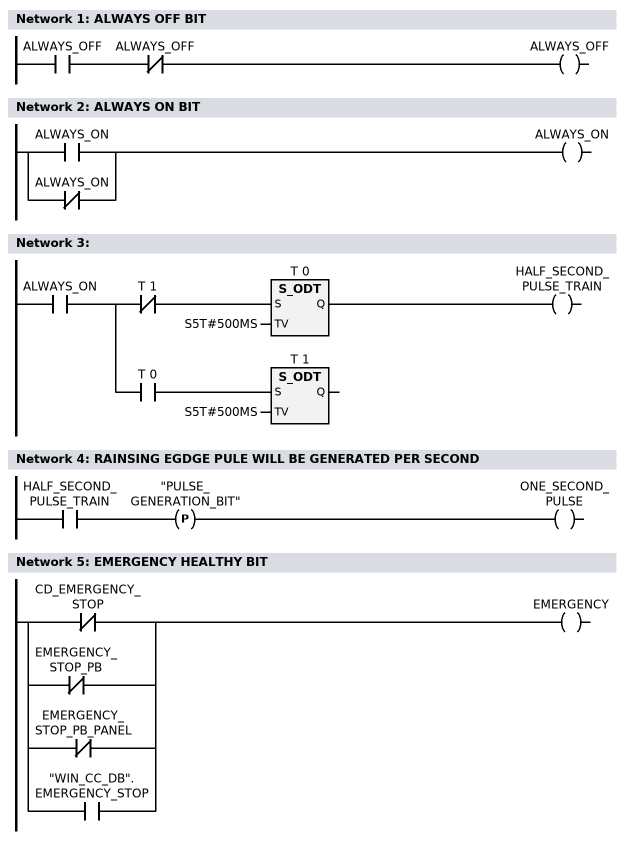
NETWORK
TITLE = ALWAYS OFF BIT
      A     "ALWAYS_OFF";
      AN    "ALWAYS_OFF";
      =     "ALWAYS_OFF";
NETWORK
TITLE = ALWAYS ON BIT
      O     "ALWAYS_ON";
      ON    "ALWAYS_ON";
      =     "ALWAYS_ON";
NETWORK
TITLE =
      A     "ALWAYS_ON";
      =     L 20.0;
      A     L 20.0;
      AN    T 1;
      L     S5T#500MS;
      SD    T 0;
      NOP   0;
      NOP   0;
      NOP   0;
      A     T 0;
      =     "HALF_SECOND_PULSE_TRAIN";
      A     L 20.0;
      A     T 0;
      L     S5T#500MS;
      SD    T 1;
      NOP   0;
      NOP   0;
      NOP   0;
      NOP   0;
NETWORK
TITLE = RAINSING EGDGE PULE WILL BE GENERATED PER SECOND
      A     "HALF_SECOND_PULSE_TRAIN";
      FP    "PULSE_GENERATION_BIT";
      =     "ONE_SECOND_PULSE";
NETWORK
TITLE = EMERGENCY HEALTHY BIT
//M0.4 LOW MEANS EMERGENCY PB NOT PRESSED.HEALTHY CONDITION
      ON    "CD_EMERGENCY_STOP";
      ON    "EMERGENCY_STOP_PB";
      ON    "EMERGENCY_STOP_PB_PANEL";
      O     "WIN_CC_DB".EMERGENCY_STOP;
      =     "EMERGENCY";
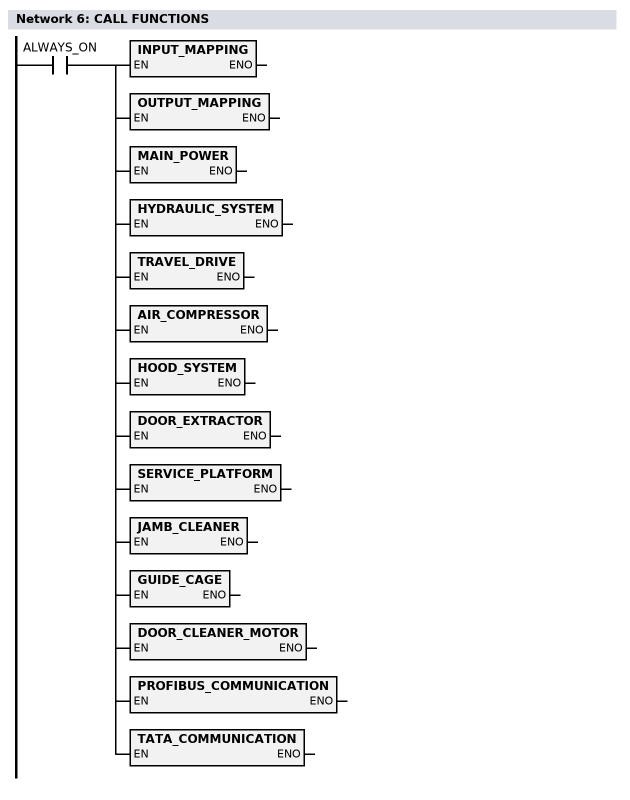
NETWORK
TITLE = CALL FUNCTIONS
      A     "ALWAYS_ON";
      =     L 20.0;
      A     L 20.0;
      JNB   _001;
      CALL  "INPUT_MAPPING";
_001: NOP   0;
      A     L 20.0;
      JNB   _002;
      CALL  "OUTPUT_MAPPING";
_002: NOP   0;
      A     L 20.0;
      JNB   _003;
      CALL  "MAIN_POWER";
_003: NOP   0;
      A     L 20.0;
      JNB   _004;
      CALL  "HYDRAULIC_SYSTEM";
_004: NOP   0;
      A     L 20.0;
      JNB   _005;
      CALL  "TRAVEL_DRIVE";
_005: NOP   0;
      A     L 20.0;
      JNB   _006;
      CALL  "AIR_COMPRESSOR";
_006: NOP   0;
      A     L 20.0;
      JNB   _007;
      CALL  "HOOD_SYSTEM";
_007: NOP   0;
      A     L 20.0;
      JNB   _008;
      CALL  "DOOR_EXTRACTOR";
_008: NOP   0;
      A     L 20.0;
      JNB   _009;
      CALL  "SERVICE_PLATFORM";
_009: NOP   0;
      A     L 20.0;
      JNB   _00a;
      CALL  "JAMB_CLEANER";
_00a: NOP   0;
      A     L 20.0;
      JNB   _00b;
      CALL  "GUIDE_CAGE";
_00b: NOP   0;
      A     L 20.0;
      JNB   _00c;
      CALL  "DOOR_CLEANER_MOTOR";
_00c: NOP   0;
      A     L 20.0;
      JNB   _00d;
      CALL  "PROFIBUS_COMMUNICATION";
_00d: NOP   0;
      A     L 20.0;
      JNB   _00e;
      CALL  "TATA_COMMUNICATION";
_00e: NOP   0;
END_ORGANIZATION_BLOCK

ORGANIZATION_BLOCK "I/O_FLT1"	// OB 82
TITLE = "I/O Point Fault"
AUTHOR : Kamillas
VERSION : 0.1
VAR_TEMP
  OB82_EV_CLASS : BYTE ;	//16#39, Event class 3, Entering event state, Internal fault event
  OB82_FLT_ID : BYTE ;	//16#XX, Fault identifcation code
  OB82_PRIORITY : BYTE ;	//Priority of OB Execution
  OB82_OB_NUMBR : BYTE ;	//82 (Organization block 82, OB82)
  OB82_RESERVED_1 : BYTE ;	//Reserved for system
  OB82_IO_FLAG : BYTE ;	//Input (01010100), Output (01010101)
  OB82_MDL_ADDR : WORD ;	//Base address of module with fault
  OB82_MDL_DEFECT : BOOL ;	//Module defective
  OB82_INT_FAULT : BOOL ;	//Internal fault
  OB82_EXT_FAULT : BOOL ;	//External fault
  OB82_PNT_INFO : BOOL ;	//Point information
  OB82_EXT_VOLTAGE : BOOL ;	//External voltage low
  OB82_FLD_CONNCTR : BOOL ;	//Field wiring connector missing
  OB82_NO_CONFIG : BOOL ;	//Module has no configuration data
  OB82_CONFIG_ERR : BOOL ;	//Module has configuration error
  OB82_MDL_TYPE : BYTE ;	//Type of module
  OB82_SUB_MDL_ERR : BOOL ;	//Sub-Module is missing or has error
  OB82_COMM_FAULT : BOOL ;	//Communication fault
  OB82_MDL_STOP : BOOL ;	//Module is stopped
  OB82_WTCH_DOG_FLT : BOOL ;	//Watch dog timer stopped module
  OB82_INT_PS_FLT : BOOL ;	//Internal power supply fault
  OB82_PRIM_BATT_FLT : BOOL ;	//Primary battery is in fault
  OB82_BCKUP_BATT_FLT : BOOL ;	//Backup battery is in fault
  OB82_RESERVED_2 : BOOL ;	//Reserved for system
  OB82_RACK_FLT : BOOL ;	//Rack fault, only for bus interface module
  OB82_PROC_FLT : BOOL ;	//Processor fault
  OB82_EPROM_FLT : BOOL ;	//EPROM fault
  OB82_RAM_FLT : BOOL ;	//RAM fault
  OB82_ADU_FLT : BOOL ;	//ADU fault
  OB82_FUSE_FLT : BOOL ;	//Fuse fault
  OB82_HW_INTR_FLT : BOOL ;	//Hardware interupt input in fault
  OB82_RESERVED_3 : BOOL ;	//Reserved for system
  OB82_DATE_TIME : DATE_AND_TIME ;	//Date and time OB82 started
END_VAR
BEGIN
// (block stored without names or comments; labels and parameter names are numbered)
END_ORGANIZATION_BLOCK

ORGANIZATION_BLOCK "RACK_FLT"	// OB 86
TITLE = "Loss Of Rack Fault"
AUTHOR : Kamillas
VERSION : 0.1
VAR_TEMP
  OB86_EV_CLASS : BYTE ;	//16#38/39 Event class 3
  OB86_FLT_ID : BYTE ;	//16#C1/C4/C5, Fault identifcation code
  OB86_PRIORITY : BYTE ;	//Priority of OB Execution
  OB86_OB_NUMBR : BYTE ;	//86 (Organization block 86, OB86)
  OB86_RESERVED_1 : BYTE ;	//Reserved for system
  OB86_RESERVED_2 : BYTE ;	//Reserved for system
  OB86_MDL_ADDR : WORD ;	//Base address of IM module in rack with fault
  OB86_RACKS_FLTD : ARRAY  [0 .. 31 ] OF BOOL ;	//Racks in fault
  OB86_DATE_TIME : DATE_AND_TIME ;	//Date and time OB86 started
END_VAR
BEGIN
// (block stored without names or comments; labels and parameter names are numbered)
END_ORGANIZATION_BLOCK

ORGANIZATION_BLOCK "PROG_ERR"	// OB 121
TITLE = "Programming Error"
AUTHOR : Kamillas
VERSION : 0.1
VAR_TEMP
  OB121_EV_CLASS : BYTE ;	//16#25, Event class 2, Entering event state, Internal fault event
  OB121_SW_FLT : BYTE ;	//16#XX Software programming fault
  OB121_PRIORITY : BYTE ;	//Priority of OB Execution
  OB121_OB_NUMBR : BYTE ;	//121 (Organization block 121, OB121)
  OB121_BLK_TYPE : BYTE ;	//16#88/8A/8B/8C/8E Type of block fault occured in
  OB121_RESERVED_1 : BYTE ;	//Reserved for system
  OB121_FLT_REG : WORD ;	//16#XX Specific register that caused fault
  OB121_BLK_NUM : WORD ;	//Number of block that programming fault occured in
  OB121_PRG_ADDR : WORD ;	//Address in block where programming fault occured
  OB121_DATE_TIME : DATE_AND_TIME ;	//Date and time OB121 started
END_VAR
BEGIN
// (block stored without names or comments; labels and parameter names are numbered)
END_ORGANIZATION_BLOCK

ORGANIZATION_BLOCK "MOD_ERR"	// OB 122
TITLE = "Module Access Error"
AUTHOR : Kamillas
VERSION : 0.1
VAR_TEMP
  OB122_EV_CLASS : BYTE ;	//16#29, Event class 2, Entering event state, Internal fault event
  OB122_SW_FLT : BYTE ;	//16#XX Software error code
  OB122_PRIORITY : BYTE ;	//Priority of OB Execution
  OB122_OB_NUMBR : BYTE ;	//122 (Organization block 122, OB122)
  OB122_BLK_TYPE : BYTE ;	//16#88/8C/8E Type of block fault occured in
  OB122_MEM_AREA : BYTE ;	//Memory area where access error occured
  OB122_MEM_ADDR : WORD ;	//Memory address where access error occured
  OB122_BLK_NUM : WORD ;	//Block number in which error occured
  OB122_PRG_ADDR : WORD ;	//Program address where error occured
  OB122_DATE_TIME : DATE_AND_TIME ;	//Date and time OB1 started
END_VAR
BEGIN
// (block stored without names or comments; labels and parameter names are numbered)
END_ORGANIZATION_BLOCK
